(* IEC 61131-3 sources: MyTestRepos/BATTERY/PRG/BATTERY, 3 files *)

(* ---- PRG_Battery.st ---- *)
PROGRAM PRG_Battery
VAR
	ManualEnterPowerSaveMode: BOOL;	(*Manual Command to enter Power Save Mode for all packs*)
	ManualExitPowerSaveMode: BOOL;	(*Manual Command to exit Power Save Mode for all packs*)

	Extended_Statemachine: UINT := 0; (*Extended state machine for IAS, containing prewarning and shutdown  *)

	M : INT; (*Master of array information in Corvus BMS*)
	P : INT; (*Pack or packs with precharge module. Must receive connect command*)

	(*Battery Commands*)
	Connect: 				BOOL; (*Connect command from state machine*)
	Disconnect: 			BOOL; (*Disconnect command from state machine*)
	Tripstatus: 			DINT; (*Trip status from state machine*)
	ConnectPack1to8: 		DINT; (* Connect command read by communication programs*)
	testPrechargeTimeout: 	BOOL; (* Used to test precharge timeout *)
	ResetBattery : 			INT; (*Reset flag to Corvus BMS. 1 or 0 for true and false.*)
	CorvusConnect: 			fb_BitToWord; (*Split word to decide which packs to connect	*)

	(* Select and connect packs *)
	bms_Connect_Pack1: BOOL;
	bms_Select_Pack1: BOOL;
	bms_Connect_Pack2: BOOL;
	bms_Select_Pack2: BOOL;
	bms_Connect_Pack3: BOOL;
	bms_Select_Pack3: BOOL;
	bms_Connect_Pack4: BOOL;
	bms_Select_Pack4: BOOL;
	bms_Connect_Pack5: BOOL;
	bms_Select_Pack5: BOOL;
	bms_Connect_Pack6: BOOL;
	bms_Select_Pack6: BOOL;
	bms_Connect_Pack7: BOOL;
	bms_Select_Pack7: BOOL;
	bms_Connect_Pack8: BOOL;
	bms_Select_Pack8: BOOL;
	ConnectRS: RS;
	DeSelectTOF: TOF;

	(*Battery Feedback*)
	BatteryAllConnected: 	BOOL; (*All packs are connected*)
	BatteryMinOneConnected: BOOL; (*At least one pack is connected*)
	BatteryDisconnected : 	BOOL; (*All packs are disconnected*)
	BatteryReady: 			BOOL; (*Precharge pack is ready to connect or in power save mode*)
	BatteryConnecting: 		BOOL; (*Precharge pack is currently connecting*)
	BatteryReadyConnect:	BOOL; (*Battery is ready to connect or already connected or in power save mode - start sequence allowed*)

	(*Power Save Mode*)
	BatteryPackPowerSaveArray : 		ARRAY[1..16] OF INT; 	(*Count packs in power save mode*)
	BatteryCountPowerSave : 			DWORD;		(* Check how many packs are in power save mode*)
	BatteryNumInPowerSave : 			INT; 		(*Number of packs in power save mode*)
	BatteryAllPacksSleeping: 			BOOL; 		(*All battery packs are in power save mode*)
	ExitPowerSaveMode : 				BOOL;		(*Command to exit power save mode for all packs.*)
	GoToPowerSaveModeTP : 				TP;			(*Command Pulse*)
	ExitPowerSaveModeTP : 				TP;			(*Command Pulse*)
	LastPackDisconnectedRT: 			R_TRIG;		(*Rising edge trigger to detect when battery pack is no longer connected*)
	DelayPowerSaveAfterDisconnectTOF: 	TOF; 		(*Delay after last pack disconnect before entering power save mode*)
	DelayPowerSaveAfterDisconnectFT:	F_TRIG;		(*Falling edge trigger to enter power save when timer has run out*)
	EmergencyGoToPowerSaveRT: 			R_TRIG;		(*Detect when battery protection calls for emergency power save*)
	ForceSleepMode:						BOOL;		(*Bit from *)
	EnterPowerSaveModeTP:				TP;			(*Pulse to enable power save mode to Corvus*)
	AllowPowerSaveMode:					BOOL;		(*Power Save is only allowed for packs not in Connected eller Connecting State*)
	BatteriesInPowerSaveArray:			ARRAY[1..16] OF INT;	(*Array to register packs in power save mode*)
	BatteriesNotAllowedToSleepArray:	ARRAY[1..16] OF INT;	(*Array to register packs which are not allowed to sleep*)

	(*SoH Verification Testing*)
	SoHCurrent: 				INT := 0; (* Current limit during SoH Verification Testing*)

	(*Battery Charge/Discharge control*)
	StopDischargeTOF: 					TOF;					(*Discharge limit reached - limit discharge current to zero for some time*)
	StopChargeTOF: 						TOF;					(*Charge limit reached - limit charge current to zero for some time*)
	BMS_DischargeLimit_eng: 			DINT := 0;				(*Current limit in ampere*)
	BMS_ChargeLimit_eng: 				DINT := 0;				(*Current limit in ampere*)
	Battery_Current_Limiter: 	fb_CorvusOrcaCurrentLimiter;	(*Limitation function based on current*)
	ChargeLimitFilter:					FILTER_I;				(*Current filter used when stopping normally*)
	DischargeLimitFilter:				FILTER_I;				(*Current filter used when stopping normally*)
	ChargeLimit_eng: 					REAL := 0;				(* Charge limit in in ampere*)
	DischargeLimit_eng: 				REAL := 0;				(* Discharge limit in in ampere*)
	DriveDischargeLimit_eng: 			REAL := 0;				(* Discharge current in ampere used to limit DC/DC drive*)
	DriveChargeLimit_eng: 				REAL := 0;				(* Charge current in ampere used to limit DC/DC drive*)

	(*Readings and statuses*)
	SoC_Floor : INT; (*Current SoC level where the batteries are disconnected due to safety reasons / undervoltage*)
	busPower: REAL := 0; (* Power in kW to/from the batteries*)
	packSOH: ARRAY [1..16] OF REAL; (*Array of all pack's State of Health*)
	packSOC: ARRAY [1..16] OF REAL; (*Array of all pack's State of Charge*)

	MinutesRemaining: REAL := 0; (*Minutes remaining till current SoC_Floor, i.e. when batteries will auto disconnect. SoC Floor can vary depending on mode.*)
	hoursRemaining: REAL := 0; (*Hours remaining till current SoC_Floor, i.e. when batteries will auto disconnect. SoC Floor can vary depending on mode.*)
	energyRemaining: REAL := 0; (*Energy remaining on batteries in kWh*)
	energyRemainingOffline: REAL := 0; (*Energy in kWh remaining on batteries in offline mode. The lowest SoC is used.*)
	EnergyToFull: REAL := 0; (*Energy in kWh remaining until fully charged, SoC = 100% *)
	EnergyToDisconnect: REAL := 0; (*Energy in kWh remaining until completely discharged, SoC = 0% *)
	batteryCharging: BOOL; (*True if current is positive, i.e. current is flowing into the batteries*)

	(*Counter variables*)
	i:INT;
	y:INT;

	(*IAS Calculated variables*)
	avgCellVolt_sum: REAL := 0;
	avgCellTemp_sum: REAL := 0;
	AvailablePower : UINT;
	avgCellVolt : INT;
	avgCellTemp : INT;
	cellBalancingStatus : ARRAY[1..16] OF BOOL;
	CellsInBalance : ARRAY[1..16] OF BOOL;
	connectionArray : ARRAY[1..16] OF BOOL;
	AvailableEnergy : UINT;
END_VAR

(*
 * =======================================================================================================================================
 * Initial paper work; select Master and map commands from state machine
 * =======================================================================================================================================
*)

(*Decide which Corvus Controller to use as (M)aster for array data and (P)recharge/connect commands*)
M := PRG_BatteryComm.M;
P := PRG_BatteryComm.P;

(*Read commands from prg_Statemachine*)
Connect := PRG_StateMain.ConnectBattery ;
Disconnect := PRG_StateMain.DisconnectBattery ;
Tripstatus := PRG_StateMain.tripStatus ;

(*
 * =======================================================================================================================================
 * Connect and Disconnect Commands
 * =======================================================================================================================================
*)

(*RS function to hold connect command to Corvus.  *)
ConnectRS(SET := (Connect AND NOT testPrechargeTimeout), RESET1 := Disconnect OR (Tripstatus <> 0));

bms_Connect_Pack1 := (PRG_HMI.setup_Battery_total_nr_of_packs >= 1) AND ConnectRS.Q1;
bms_Connect_Pack2 := (PRG_HMI.setup_Battery_total_nr_of_packs >= 2) AND ConnectRS.Q1;
bms_Connect_Pack3 := (PRG_HMI.setup_Battery_total_nr_of_packs >= 3) AND ConnectRS.Q1;
bms_Connect_Pack4 := (PRG_HMI.setup_Battery_total_nr_of_packs >= 4) AND ConnectRS.Q1;
bms_Connect_Pack5 := (PRG_HMI.setup_Battery_total_nr_of_packs >= 5) AND ConnectRS.Q1;
bms_Connect_Pack6 := (PRG_HMI.setup_Battery_total_nr_of_packs >= 6) AND ConnectRS.Q1;
bms_Connect_Pack7 := (PRG_HMI.setup_Battery_total_nr_of_packs >= 7) AND ConnectRS.Q1;
bms_Connect_Pack8 := (PRG_HMI.setup_Battery_total_nr_of_packs >= 8) AND ConnectRS.Q1;

DeSelectTOF(
		IN := ConnectRS.Q1,
		PT := T#2500ms
);

(*Make sure packs are not de-selected prior to disconnect command*)
bms_Select_Pack1 := DeSelectTOF.Q;
bms_Select_Pack2 := DeSelectTOF.Q;
bms_Select_Pack3 := DeSelectTOF.Q;
bms_Select_Pack4 := DeSelectTOF.Q;
bms_Select_Pack5 := DeSelectTOF.Q;
bms_Select_Pack6 := DeSelectTOF.Q;
bms_Select_Pack7 := DeSelectTOF.Q;
bms_Select_Pack8 := DeSelectTOF.Q;

(*Prepare connection setup to Corvus*)
CorvusConnect(
	EN := TRUE,
	Bit0 := bms_Connect_Pack1,
	Bit1 := bms_Select_Pack1,
	Bit2 := bms_Connect_Pack2,
	Bit3 := bms_Select_Pack2,
	Bit4 := bms_Connect_Pack3,
	Bit5 := bms_Select_Pack3,
	Bit6 := bms_Connect_Pack4,
	Bit7 := bms_Select_Pack4,
	Bit8 := bms_Connect_Pack5,
	Bit9 := bms_Select_Pack5,
	Bit10 := bms_Connect_Pack6,
	Bit11 := bms_Select_Pack6,
	Bit12 := bms_Connect_Pack7,
	Bit13 := bms_Select_Pack7,
	Bit14 := bms_Connect_Pack8,
	Bit15 := bms_Select_Pack8,
	OUT => ConnectPack1to8
);

(*Battery is connected only when all packs are connected*)
BatteryAllConnected := (PRG_BatteryComm.CorvusRead[M].theArray.nrOfPackConnected = PRG_HMI.setup_Battery_total_nr_of_packs);

(*At least one pack is connected*)
BatteryMinOneConnected := (PRG_BatteryComm.CorvusRead[M].theArray.nrOfPackConnected >= 1);

(*Battery is disconnected only when all packs are disconnected*)
BatteryDisconnected := (PRG_BatteryComm.CorvusRead[M].theArray.nrOfPackConnected = 0);

(*Battery is ready when Pack controller with precharge is ready*)
BatteryReady := ((PRG_BatteryComm.CorvusRead[P].Pack.operationMode = 3) OR (PRG_BatteryComm.CorvusRead[P].Pack.operationMode = 1));

(*Connecting when precharge pack is working its magic*)
BatteryConnecting := (PRG_BatteryComm.CorvusRead[P].Pack.operationMode = 4);

(*Battery Ready to be Connected*)
BatteryReadyConnect := ((PRG_BatteryComm.CorvusRead[P].Pack.operationMode = 3) OR (PRG_BatteryComm.CorvusRead[P].Pack.operationMode = 5) OR (PRG_BatteryComm.CorvusRead[P].Pack.operationMode = 1));

(*
 * =======================================================================================================================================
 * Power Save Mode
 * =======================================================================================================================================
*)

(*Protection conditions to enter power save mode*)
EmergencyGoToPowerSaveRT(CLK := ForceSleepMode);

(*Enter power save mode when disconnect timer has run out*)
LastPackDisconnectedRT(
	CLK := (NOT BatteryMinOneConnected),
);

(*Enter power save mode when disconnect timer has run out*)
DelayPowerSaveAfterDisconnectTOF(
	IN := LastPackDisconnectedRT.Q,
	PT := REAL_TO_TIME(PRG_HMI.Delay_EnterPowerSaveMode*3600000)
);
DelayPowerSaveAfterDisconnectFT(CLK:=DelayPowerSaveAfterDisconnectTOF.Q);

EnterPowerSaveModeTP(
	IN := (DelayPowerSaveAfterDisconnectFT.Q OR ManualEnterPowerSaveMode OR EmergencyGoToPowerSaveRT.Q) AND PRG_HMI.enPowerSaveMode AND AllowPowerSaveMode,
	PT := T#2s,
	Q => (*Output is read in PRG_BatteryComm*),
	ET =>
);

(*Exit power save mode when starting*)
ExitPowerSaveModeTP(
	IN := PRG_Operation.ControlPlace.Start OR ManualExitPowerSaveMode,
	PT := T#2s,
	Q => ExitPowerSaveMode,
	ET =>
);

(*For loop to check how the batteries are sleeping or if they are allowed to go to sleep*)
FOR i:=1 TO PRG_HMI.setup_Battery_total_nr_of_packs BY 1 DO

	(*Check which batteries are in power save mode*)
	IF (PRG_BatteryComm.CorvusRead[i].Pack.operationMode = 1) THEN
		BatteriesInPowerSaveArray[i] := i*1;
	ELSE
		BatteriesInPowerSaveArray[i] := 0;
	END_IF

	(*Check which batteries are not allowed to enter power save*)
	IF (PRG_BatteryComm.CorvusRead[i].Pack.operationMode = 4 OR PRG_BatteryComm.CorvusRead[i].Pack.operationMode = 5) THEN
		BatteriesNotAllowedToSleepArray[i] := i*1;
	ELSE
		BatteriesNotAllowedToSleepArray[i] := 0;
	END_IF

END_FOR

(*Check how many battery packs are in power save mode*)
BatteryNumInPowerSave :=	BIT_COUNT(REAL_TO_DWORD((ARRAY_SUM(pt := ADR(BatteriesInPowerSaveArray), size := SIZEOF(BatteriesInPowerSaveArray)))));
IF (BatteryNumInPowerSave = PRG_HMI.setup_Battery_total_nr_of_packs) THEN
	BatteryAllPacksSleeping := TRUE;
ELSE
	BatteryAllPacksSleeping := FALSE;
END_IF

(*Power Save Mode is not allowed if any pack is either connected or connected*)
AllowPowerSaveMode := ( ARRAY_MAX(pt := ADR(BatteriesNotAllowedToSleepArray), size := SIZEOF(BatteriesNotAllowedToSleepArray))   <> 0);

(*
 * =======================================================================================================================================
 * Limitation of power to and from battery
 * =======================================================================================================================================
*)

(*------------------------------------- Batterilimiter fra BMS----------------------------------------------*)
(*This logic alters current limiters being sent into the limiter block. The output is filtered and controlled to vacon*)
IF (PRG_HMI.ChargeDischargeCurrentTestActive) THEN
	BMS_ChargeLimit_eng := LIMIT (0,REAL_TO_DINT(PRG_HMI.ChargeCurrentLimit_scale.PV),PRG_BatteryComm.CorvusRead[M].theArray.systemChargelimit);
	BMS_DischargeLimit_eng := LIMIT (0,REAL_TO_DINT(PRG_HMI.DischargeCurrentLimit_scale.PV),PRG_BatteryComm.CorvusRead[M].theArray.systemDischargeLimit);

ELSIF (PRG_HMI.SoHVerifModeActive) THEN (*Limit current to C-rate during State of Health Verification testing*)
	BMS_ChargeLimit_eng := LIMIT (0,INT_TO_DINT(SoHCurrent),PRG_BatteryComm.CorvusRead[M].theArray.systemChargelimit);
	BMS_DischargeLimit_eng := LIMIT (0,INT_TO_DINT(SoHCurrent),PRG_BatteryComm.CorvusRead[M].theArray.systemDischargeLimit);

ELSE
	BMS_ChargeLimit_eng := PRG_BatteryComm.CorvusRead[M].theArray.systemChargelimit;
	BMS_DischargeLimit_eng := PRG_BatteryComm.CorvusRead[M].theArray.systemDischargeLimit;
END_IF

(*Reading Charge/discharge limits and bus current in Ampere from BMS and compensates it by manipulating the reference*)
Battery_Current_Limiter(
	BMS_ChargeLimit_in := DINT_TO_INT(BMS_ChargeLimit_eng),
	BMS_DischargeLimit_in := DINT_TO_INT(BMS_DischargeLimit_eng),
	BatteryCurrent := PRG_BatteryComm.CorvusRead[M].theArray.busCurrent,
	NominalDriveCurrent := PRG_HMI.DriveSettings.SourceNomCurrent,
	BatteryConnected := BatteryMinOneConnected,
	ChargeLimit_eng => ,
	DischargeLimit_eng => ,
	ChargingLimited => ,
	DischargingLimited =>
);

(*Stop charging when battery voltage or SoC is too high*)
StopChargeTOF(
	IN := PRG_BatteryProtection.ChargeLimitWord <> 0,
	PT := T#30s, (*We want to stop charging for at least some time to prevent "blinking" of limits*)
	Q => ,
	ET =>
);

 (*Stop discharging when battery voltage or SoC is too low*)
StopDischargeTOF(
	IN:= PRG_BatteryProtection.DischargeLimitWord <> 0,
	PT := T#30s, (*We want to stop charging for at least some time to prevent "blinking" of limits*)
	Q => ,
	ET =>
);

(*Calculate charge/discharge limit from C-rate - Used as input to BMS Limiter during SoH verification*)
SoHCurrent := REAL_TO_INT(PRG_HMI.SoHChargeDischargeRate * setup_Battery_C_Rate * PRG_BatteryComm.CorvusRead[M].theArray.nrOfPackConnected);

(*This logic alters limits. Used for deloading or limiting when past SoC Low and Soc High*)

(*Ramping down limits towards zero to deload when stopping*)
IF ((PRG_StateMain.State = e_Stopping))  THEN
	ChargeLimit_eng := 0;
	DischargeLimit_eng := 0;

(*Limit when over charging - allowed to discharge*)
ELSIF (StopChargeTOF.Q) THEN
	ChargeLimit_eng := 0;
	DischargeLimit_eng := Battery_Current_Limiter.DischargeLimit_eng;

(*Limit when over discharging - allowed to charge*)
ELSIF (StopDischargeTOF.Q) THEN
	ChargeLimit_eng := Battery_Current_Limiter.ChargeLimit_eng;
	DischargeLimit_eng :=	0;

(*Normal operational limits controlled by BMS and other protective functions*)
ELSE
	ChargeLimit_eng := 		Battery_Current_Limiter.ChargeLimit_eng;
	DischargeLimit_eng := 	Battery_Current_Limiter.DischargeLimit_eng;
END_IF

(* Filtering of limit value*)
DischargeLimitFilter(
	X := REAL_TO_INT(DischargeLimit_eng),
	T := T#2s
);

ChargeLimitFilter(
	X := REAL_TO_INT(ChargeLimit_eng),
	T := T#2s
);

(*Preparing limit value to PRG_Drive*)
DriveChargeLimit_eng := 		ChargeLimitFilter.Y;
DriveDischargeLimit_eng := 		DischargeLimitFilter.Y;

(*
 * =======================================================================================================================================
 * Calculate Energy in batteries and time to full/empty/disconnect
 * =======================================================================================================================================
*)

(* Check if we are charging or discharging the battery *)
batteryCharging := (PRG_BatteryComm.CorvusRead[M].theArray.busPowerCalculated > 0 AND (PRG_BatteryComm.CorvusRead[M].Pack.operationMode = 5));

(*Calculate offline available energy, based on all packs and minimum state of charge*)
energyRemainingOffline := (
 	ARRAY_MIN(pt:=ADR(packSOC), size:=SIZEOF(packSOC)) *  	(* Lowest State of Charge *)
	setup_Energy_per_pack *									(* kWh per pack *)
	PRG_HMI.setup_Battery_total_nr_of_packs *				(* Total number of packs in array *)
	ARRAY_MIN(pt:=ADR(packSOH), size:=SIZEOF(packSOH)) *	(* Systems state of health *)
	0.0001													(* Correction factor *)
);

(*Calculate remaining energy to zero in an online system*)
EnergyToDisconnect := (
 	(PRG_BatteryComm.CorvusRead[M].theArray.systemOnlineSOC - REAL_TO_DINT(PRG_HMI.BMS_SoC.LL)) *  (* State of charge *)
	setup_Energy_per_pack *											(* kWh per pack *)
	PRG_BatteryComm.CorvusRead[M].theArray.nrOfPackConnected *		(* Number of packs online *)
	PRG_BatteryComm.CorvusRead[M].theArray.systemOnlineSOH *		(* Systems state of health *)
	0.0001															(* Correction factor *)
);

(*Calculate energy to full state of charge in an online system*)
EnergyToFull := (
 	setup_Energy_per_pack * 										(* kWh per pack *)
 	PRG_BatteryComm.CorvusRead[M].theArray.nrOfPackConnected *		(* Number of packs online *)
	PRG_BatteryComm.CorvusRead[M].theArray.systemOnlineSOH *		(* Systems state of health *)
	0.01															(* Correction factor *)
) - EnergyToDisconnect;												(* Subtract remaining energy *)

(*Prevent division by zero when calculating time remaining (This result is the denominator in the energy division) *)
IF PRG_BatteryComm.CorvusRead[M].theArray.busPowerCalculated = 0
	THEN busPower := 0.1;
	ELSE busPower := PRG_BatteryComm.CorvusRead[M].theArray.busPowerCalculated;
END_IF

(* Calculate time remaining to either 100% or 0% depending on whether the battery is charging or discharging *)
IF (batteryCharging) THEN
	hoursRemaining := EnergyToFull/busPower;
ELSE
	hoursRemaining := EnergyToDisconnect/busPower;
END_IF

MinutesRemaining := ABS(hoursRemaining*60);

(*
 * =======================================================================================================================================
 * Calculate values for IAS information
 * =======================================================================================================================================
*)

FOR i:=1 TO 16 BY 1 DO

	(*Set up all pack state of charges in an array*)
	IF ((PRG_BatteryComm.CorvusRead[i].Pack.SOC <> 0) OR PRG_BatteryComm.CorvusRead[i].ModbusFault) THEN
		packSOC[i] := DINT_TO_REAL(PRG_BatteryComm.CorvusRead[i].Pack.SOC);
	ELSE
		packSOC[i] := 999; (*prevent zeros in array when looking for the lowest value*)
	END_IF

	(*Set up all pack state of health in an array*)
	IF ((PRG_BatteryComm.CorvusRead[i].Pack.SOH <> 0) OR PRG_BatteryComm.CorvusRead[i].ModbusFault) THEN
		packSOH[i] := DINT_TO_REAL(PRG_BatteryComm.CorvusRead[i].Pack.SOH);
	ELSE
		packSOH[i] := 999; (*prevent zeros in array when looking for the lowest value*)
	END_IF

	(*Count pack balancing status*)
	IF (PRG_BatteryComm.CorvusRead[i].Pack.cellBalancingStatus = 1) THEN
		cellBalancingStatus[i] :=  TRUE;
	ELSE
		cellBalancingStatus[i] :=  FALSE;
	END_IF;

	(*Count pack balancing status 2*)
	IF (PRG_BatteryComm.CorvusRead[i].Pack.cellsInBalance = 1) THEN
		CellsInBalance[i] :=  TRUE;
	ELSE
		CellsInBalance[i] :=  FALSE;
	END_IF;

	(*Connection Array*)
	IF (PRG_BatteryComm.CorvusRead[i].Pack.operationMode = 5) THEN
		connectionArray[i] :=  TRUE;
	ELSE
		connectionArray[i] :=  FALSE;
	END_IF;
END_FOR

(*Find average cell temperature*)
avgCellTemp_sum := 0;
FOR i:=1 TO PRG_HMI.setup_Battery_total_nr_of_packs BY 1 DO
	avgCellTemp_sum := avgCellTemp_sum + DINT_TO_REAL(PRG_BatteryComm.CorvusRead[i].Pack.avgCellTemp);
END_FOR
avgCellTemp := REAL_TO_INT(fun_SafeDivide(divident := avgCellTemp_sum, devisor := PRG_HMI.setup_Battery_total_nr_of_packs));

(*Find average cell voltage*)
avgCellVolt_sum := 0;
FOR i:=1 TO PRG_HMI.setup_Battery_total_nr_of_packs BY 1 DO
	avgCellVolt_sum := avgCellVolt_sum + DINT_TO_REAL(PRG_BatteryComm.CorvusRead[i].Pack.avgCellVoltage);
END_FOR
avgCellVolt := REAL_TO_INT(fun_SafeDivide(divident := avgCellVolt_sum, devisor := PRG_HMI.setup_Battery_total_nr_of_packs));

(*Determine wether to use online or offline energy*)
IF (PRG_BatteryComm.CorvusRead[M].theArray.nrOfPackConnected > 0) THEN
	AvailableEnergy := REAL_TO_UINT(EnergyToDisconnect);
ELSE
	AvailableEnergy := REAL_TO_UINT(energyRemainingOffline);
END_IF

(*Send offline estimated available power to IAS/PMS*)
IF (PRG_BatteryComm.CorvusRead[M].theArray.nrOfPackConnected > 0) THEN
	AvailablePower := REAL_TO_UINT( MIN(PRG_BatteryComm.CorvusRead[M].theArray.systemDischargeLimit,PRG_HMI.DriveSettings.SourceNomCurrent) * PRG_BatteryComm.CorvusRead[M].theArray.busVoltage/1000);
ELSE
	AvailablePower := REAL_TO_UINT((PRG_HMI.DriveSettings.SourceNomCurrent * PRG_BatteryComm.CorvusRead[M].Pack.batteryVoltage)/1000);
END_IF

(* IAS extended state machine status containing prewarning and shutdown *)
IF (PRG_BatteryProtection.batteryPreWarning AND NOT (PRG_StateMain.tripStatus <> 0)) THEN
	Extended_Statemachine := 6;
ELSIF (PRG_StateMain.tripStatus <> 0) THEN
	Extended_Statemachine := 7;
ELSE
	Extended_Statemachine := PRG_StateMain.State;;
END_IF

END_PROGRAM

ACTIONS

END_ACTIONS

(* ---- PRG_BatteryComm.st ---- *)
(*
 * This program instantiates the Corvus Orca communication function block and gathers write-commands from other programs.
 * Made by: YS
 * Last changed: 2018-09-18
*)
PROGRAM PRG_BatteryComm

VAR
	mb_BMS_arrayData: 	ARRAY [1..16] OF str_Corvus_Array; 		(*Almighty array containing all information about PV and alarms for analog input signals*)
	mb_BMS_packData: 	ARRAY [1..16] OF str_Corvus_packData;	(*Almighty array containing all information about PV and alarms for analog input signals*)
	mb_BMS_packFW: 		ARRAY [1..16] OF str_Corvus_packFW; 	(*Almighty array containing all information about PV and alarms for analog input signals*)
    CorvusRead: 		ARRAY [1..16] OF str_Corvus_ALL; 		(*The almighty Corvus BMS Array-Array*)
	CorvusWrite: 		ARRAY [1..16] OF str_Corvus_Write;		(*Command Register Array to Corvus pack controllers*)

	CorvusModbusFault_TON: 				TON;							(*Timer to declare modbus communication fault*)
	Modbus_Wait:						BOOL;							(*Start to wait before restarting modbus fault checking*)
	Modbus_WaitRT:						R_TRIG;							(*Puls detection to start timer*)
	Modbus_WaitTryFT:					F_TRIG;							(*Puls detection that timer has ended*)
	ModbusFault_WaitTry_TP:				TP;								(*Timer to wait before restarting check of array*)
	CorvusBMS_Total_Comm_Fault_SR:		SR;								(*The Total Modbus Fault must be latched unntil we know it is healthy again*)
	CorvusBMS_Reset_Total_Comm_Fault_TON:TON;							(*Wait this long before declaring that communication is OK again*)
	NoPrechargePackComm: 				BOOL; 							(*Alarm when there is modbus fault on all packs which can start/stop*)
	n: 									INT := 0; 						(*Looping variable for reset function*)
	i: 									INT; 							(*Looping variable for checking comm fault across packs*)
	M : 								INT:=1; 						(*Pack number for current Array Master: The pack that array information is gathered from*)
	P : 								INT:=1; 						(*Pack number for current Array Precharge Master: The pack that can initiate start/connect requests*)
	Corvus_Array : 						fb_CorvusOrcaComm; 				(*All corvus data*)
	WriteCommands : 					ARRAY[1..16] OF str_Corvus_Write; (*Command Register Array to Corvus pack controllers*)

	(*Commands read from other programs*)
	Reset : 							BOOL; 							(*Reset command for battery packs*)
	CorvusBMS_Total_Comm_Fault_TON : 	TON;
	CorvusBMS_Total_Comm_Fault: 		BOOL; 							(*No communication with any Corvus batteries :( *)

	(*Variables to HMI*)
	setup_AlarmDelay_Modbus : 			TIME:=T#5s;		(*Delay before issuing total comm failure alarm*)
END_VAR

Reset := PRG_Functions.Reset;

(*
 * =======================================================================================================================================
 * Communication with Corvus Orca Battery Management
 * =======================================================================================================================================
*)
Corvus_Array(
 	First_Card_ID:=PRG_HMI.setup_Battery_First_Card_Nr,
 	Number_of_packs_in_array:=PRG_HMI.setup_Battery_total_nr_of_packs ,
 	corvusWrite := WriteCommands,
 	Reset := Reset,
 	output => CorvusRead
);

(*
 * =======================================================================================================================================
 * Find Array Master (M) - This is the array we use most data from
 * =======================================================================================================================================
*)

IF CorvusRead[M].ModbusFault AND CorvusRead[1].ModbusFault AND  M<= PRG_HMI.setup_Battery_total_nr_of_packs AND NOT ModbusFault_WaitTry_TP.Q  THEN
	(*If current array master and pack 1 has comm fault, try next one as long as we still have more packs in the array to try*)
	M := M+1;
	Modbus_Wait := FALSE;
ELSIF M > PRG_HMI.setup_Battery_total_nr_of_packs OR NOT CorvusRead[1].ModbusFault THEN
	(*If array 1 is ok *OR* there are no more arrays to try - go for number 1*)
	M := 1;
	Modbus_Wait := TRUE;	(*After running through all arrays, wait before restarting so that CorvusBMS_Total_Comm_Fault_TON can detect that we have no-one to talk to*)
END_IF

Modbus_WaitRT(CLK := Modbus_Wait); (*Create an R_trig to start the TP*)
ModbusFault_WaitTry_TP(				(*When we have tested all arrays and found no-one to communicate with, take a pause before re-starting so that we can detect the comm fault*)
		IN := Modbus_WaitRT.Q,
		PT := setup_AlarmDelay_Modbus + INT_TO_TIME(1000) (*Make sure that the re-try delay is longer than the alarm delay. 1000 = 1 s *)
	);
Modbus_WaitTryFT(CLK := ModbusFault_WaitTry_TP.Q); (*Detect when the pause is finished so that the pause-command can be turned off*)

IF(Modbus_WaitTryFT.Q OR NOT CorvusRead[M].ModbusFault) THEN
	Modbus_Wait := FALSE;
END_IF

(*No success in finding an Array master without communication fault - issue alarm*)
CorvusBMS_Total_Comm_Fault_TON(
	IN := CorvusRead[M].ModbusFault,
	PT := setup_AlarmDelay_Modbus
);

(*Make sure that the re-established communication is stable before clearing the alarm*)
CorvusBMS_Reset_Total_Comm_Fault_TON(
	IN := NOT Modbus_Wait,
	PT := setup_AlarmDelay_Modbus + INT_TO_TIME(2000), (*The "stable time" must be longer than the pause between retry-attemps*)
	Q => ,
	ET =>
);

(*Latch the modbus fault and reset it when communication has been restored for a time*)
CorvusBMS_Total_Comm_Fault_SR(
	SET1 := CorvusBMS_Total_Comm_Fault_TON.Q,
	RESET := CorvusBMS_Reset_Total_Comm_Fault_TON.Q OR PRG_Functions.Reset,
	Q1 => CorvusBMS_Total_Comm_Fault
);

(*
 * =======================================================================================================================================
 * Find Array Precharge Master (P) - This is the array we send start commands to
 * =======================================================================================================================================
*)

IF NOT CorvusRead[setup_Battery_PrechargePackA].ModbusFault THEN
	(*If pack A is home sick but pack B is ok - it's all good*)
	P := setup_Battery_PrechargePackA;
	NoPrechargePackComm := FALSE;
ELSE
	NoPrechargePackComm := TRUE;
END_IF

(*
 * =======================================================================================================================================
 * Write Commands
 * =======================================================================================================================================
*)

(*Connect Commands*)
WriteCommands[M].connectPack1to8 := PRG_Battery.ConnectPack1to8;

(*Power Save Commands*)
IF (PRG_Battery.EnterPowerSaveModeTP.Q) THEN
	WriteCommands[M].systemPowerSaveControl := 2;
ELSIF (PRG_Battery.ExitPowerSaveModeTP.Q) THEN
	WriteCommands[M].systemPowerSaveControl := 3;
ELSE
	WriteCommands[M].systemPowerSaveControl := 0;
END_IF

(* Reset all pack controllers *)
IF (Reset AND CorvusRead[M].theArray.nrOfPackFault > 0) THEN
	FOR n := 1 TO PRG_HMI.setup_Battery_total_nr_of_packs BY 1 DO
		WriteCommands[n].systemAlarmReset := 1;
	END_FOR
	n := 1;
ELSIF(Reset AND CorvusRead[M].theArray.nrOfPackFault = 0) THEN
	FOR n := 1 TO PRG_HMI.setup_Battery_total_nr_of_packs BY 1 DO
		WriteCommands[n].systemAlarmReset := 0;
	END_FOR
	n := 1;
ELSIF(NOT Reset) THEN
	FOR n := 1 TO PRG_HMI.setup_Battery_total_nr_of_packs BY 1 DO
		WriteCommands[n].systemAlarmReset := 0;
	END_FOR
	n := 1;
END_IF

;
END_PROGRAM

ACTIONS

END_ACTIONS

(* ---- PRG_BatteryProtection.st ---- *)
PROGRAM PRG_BatteryProtection
VAR
	(* Find any BMS Array warning associated with a pre-warning*)
	batteryPreWarning: 			BOOL; 					(*True if any pack has one or more prewarning alarms*)
	BatteryPreWarnings_Array: 	ARRAY[1..16] OF INT; 	(*Array to gather information about prewarning alarms from all packs*)

	(*Find any common warning from the battery array*)
	batteryCommonWarning: 		BOOL; 					(*True if any pack has one or more warnings*)
	BatteryWarnings_Array: 		ARRAY[1..16] OF INT; 	(*Array to gather information about warning alarms from all packs*)

	(*Find any common fault from the battery array*)
	batteryCommonFault: 		BOOL; (*True if any pack has an active/unacknowledged fault*)

	(*Common Faults from Battery Array*)
	Common_SE_overVoltage_Fault_Array: 					ARRAY[1..16] OF INT; (*Array of BOOLs from BMS: *)
	Common_SE_underVoltage_Fault_Array: 				ARRAY[1..16] OF INT; (*Array of BOOLs from BMS: *)
	Common_SE_overTemperature_Fault_Array: 				ARRAY[1..16] OF INT; (*Array of BOOLs from BMS: *)
	Common_HVIL_Fault_Array: 							ARRAY[1..16] OF INT; (*Array of BOOLs from BMS: *)
	Common_E_Stop_Active_Fault_Array: 					ARRAY[1..16] OF INT; (*Array of BOOLs from BMS: *)
	Common_Safety_Shutdown_Fault_Array: 				ARRAY[1..16] OF INT; (*Array of BOOLs from BMS: *)
	Common_Ground_Fault_Fault_Array: 					ARRAY[1..16] OF INT; (*Array of BOOLs from BMS: *)
	Common_Contactor_Fault_Array: 						ARRAY[1..16] OF INT; (*Array of BOOLs from BMS: *)
	Common_Low_Temp_OverCurrent_Fault_Array: 			ARRAY[1..16] OF INT; (*Array of BOOLs from BMS: *)
	Common_Repeated_OverCharge_Lockout_Fault_Array: 	ARRAY[1..16] OF INT; (*Array of BOOLs from BMS: *)
	Common_Deep_OverDischarge_Lockout_Fault_Array: 		ARRAY[1..16] OF INT; (*Array of BOOLs from BMS: *)
	Common_PDM_OverTemperature_Fault_Array: 			ARRAY[1..16] OF INT; (*Array of BOOLs from BMS: *)

	Common_SE_overVoltage_Fault: 				BOOL; (*Any pack has a Cell Over Voltage Fault*)
	Common_SE_underVoltage_Fault: 				BOOL; (*Any pack has a Cell Under Voltage Fault*)
	Common_SE_overTemperature_Fault: 			BOOL; (*Any pack has a Cell Over Temperature Fault*)
	Common_HVIL_Fault: 							BOOL; (*Any pack has a High Voltage Interlock Loop fault*)
	Common_E_Stop_Active_Fault: 				BOOL; (*Any pack has a Emergency Stop Active Fault*)
	Common_Safety_Shutdown_Fault: 				BOOL; (*Any pack has a Safety Shutdown Fault*)
	Common_Ground_Fault_Fault: 					BOOL; (*Any pack has a Ground Fault*)
	Common_Contactor_Fault: 					BOOL; (*Any pack has a Contactor Fault*)
	Common_Low_Temp_OverCurrent_Fault: 			BOOL; (*Any pack has a Low Temperature Over Current Fault*)
	Common_Repeated_OverCharge_Lockout_Fault: 	BOOL; (*Any pack has a Repeated Over Charge Lockout Fault*)
	Common_Deep_OverDischarge_Lockout_Fault: 	BOOL; (*Any pack has a Common Deep Over Discharge Lockout Fault*)
	Common_PDM_OverTemperature_Fault: 			BOOL; (*Any pack has a Power Distribution Module Over Temperature Fault*)

	(*Common Warnings from Battery Array*)
	Common_SE_overVoltage_Warning_Array: 		ARRAY[1..16] OF INT; (*Array of BOOLs from BMS: *)
	Common_SE_underVoltage_Warning_Array: 		ARRAY[1..16] OF INT; (*Array of BOOLs from BMS: *)
	Common_SE_overTemperature_Warning_Array: 	ARRAY[1..16] OF INT; (*Array of BOOLs from BMS: *)
	Common_Module_Communication_Warning_Array: 	ARRAY[1..16] OF INT; (*Array of BOOLs from BMS: *)
	Common_OverCurrent_Warning_Array: 			ARRAY[1..16] OF INT; (*Array of BOOLs from BMS: *)
	Common_Input_PowerLoss_Warning_Array: 		ARRAY[1..16] OF INT; (*Array of BOOLs from BMS: *)
	Common_PDM_overTemperature_Warning_Array: 	ARRAY[1..16] OF INT; (*Array of BOOLs from BMS: *)
	Common_CoolantLeak_Warning_Array: 			ARRAY[1..16] OF INT; (*Array of BOOLs from BMS: *)
	Common_SE_overVoltage_Warning: 				BOOL; (*Any pack has a Common Cell Over Voltage Warning*)
	Common_SE_underVoltage_Warning: 			BOOL; (*Any pack has a Common Cell Under Voltage Warning*)
	Common_SE_overTemperature_Warning: 			BOOL; (*Any pack has a Common Cell Over Temperature Warning*)
	Common_Module_Communication_Warning: 		BOOL; (*Any pack has a Common Module Communication Warning*)
	Common_OverCurrent_Warning: 				BOOL; (*Any pack has a Common Over Current Warning*)
	Common_Input_PowerLoss_Warning: 			BOOL; (*Any pack has a Common Input Powerloss Warning*)
	Common_PDM_overTemperature_Warning: 		BOOL; (*Any pack has a Common Power Distribution Module Over Temperature Warning*)
	Common_CoolantLeak_Warning: 				BOOL; (*Any pack has a Common Coolant Water Leakage Warning*)

	CorvusRead: 			ARRAY [1..16] OF str_Corvus_ALL; (*The almighty Corvus BMS Array-Array*)
	BatteryAlone :			BOOL; 			(*If battery is alone, lower SoC trip limit is decreased*)
	BatteryCharging:	 	BOOL;			(*If battery is charging, discharging is still allowed beyond limits*)
	ConfigError:			INT;			(*Check that all protection settings are within hardcoded limits*)

	TripBasket : 			fb_16DelayedSR;	(*Collection basket for protection trips*)
	WarningBasket :			fb_16DelayedSR; (*Collection basket for warnings*)
	ProtectionTrip: 		DINT;			(*All bits from protection trips*)
	ChargeLimitWord :		WORD;			(*Word with bit-conditions for stop charging*)
	DischargeLimitWord :	WORD;			(*Word with bit-conditions for stop discharging*)

	Warning_SoC_L : 				BOOL;	(*Warning or trip bit*)
	Warning_SoC_L_Offline :			BOOL;	(*Warning or trip bit*)
	Warning_SoC_LL_Offline :		BOOL;	(*Warning or trip bit*)
	Warning_SoC_H : 				BOOL;	(*Warning or trip bit*)
	Warning_Volt_L : 				BOOL;	(*Warning or trip bit*)
	Warning_Volt_H : 				BOOL;	(*Warning or trip bit*)
	Warning_CellVolt_H :			BOOL;	(*Warning or trip bit*)
	Warning_CellVolt_L :			BOOL;	(*Warning or trip bit*)
	Warning_CellVolt_L_Offline :	BOOL;	(*Warning or trip bit*)
	Warning_CellVolt_LL_Offline :	BOOL;	(*Warning or trip bit*)
	Warning_CellTemp_H :			BOOL;	(*Warning or trip bit*)
	Warning_CellTemp_L :			BOOL;	(*Warning or trip bit*)
	Warning_BattRoomTemp_HH:		BOOL;	(*Warning or trip bit*)
	Warning_BattRoomTemp_H:			BOOL;	(*Warning or trip bit*)
	Warning_BattRoomTemp_L:			BOOL;	(*Warning or trip bit*)
	Warning_BattRoomTemp_LL:		BOOL;	(*Warning or trip bit*)

	ProtectionTrip_SoC_HH: 			BOOL;	(*Warning or trip bit*)
	ProtectionTrip_SoC_LL: 			BOOL;	(*Warning or trip bit*)
	ProtectionTrip_SoC_LLL: 		BOOL;	(*Warning or trip bit*)
	ProtectionTrip_CellTemp_HH:		BOOL;	(*Warning or trip bit*)
	ProtectionTrip_CellVolt_HH:		BOOL;	(*Warning or trip bit*)
	ProtectionTrip_CellVolt_LL:		BOOL;	(*Warning or trip bit*)
	ProtectionTrip_Overvoltage: 	BOOL;	(*Warning or trip bit*)
	ProtectionTrip_Undervoltage: 	BOOL;	(*Warning or trip bit*)
	M:INT;

	(*Offline Protection*)
	ForceSleepMode :		BOOL;					(*Conditions are so that we want to force batteries to sleep*)
	i: 						INT;					(*Looping variable*)
	minCellVoltage: 		REAL := 0;				(*The lowest cell voltage in the array*)
	minCellVoltageArray: 	ARRAY[1..16] OF REAL;	(*Array of lowest cell voltages in battery packs*)
	maxCellVoltage: 		REAL := 0;				(*The highest cell voltage in the array*)
	maxCellVoltageArray: 	ARRAY[1..16] OF REAL;	(*Array of highest cell voltages in battery packs*)

	minCellTemp: 			REAL := 0;				(*The lowest cell temperature in the array*)
	minCellTempArray: 		ARRAY[1..16] OF REAL;	(*Array of lowest cell temperature in battery packs*)
	maxCellTemp: 			REAL := 0;				(*The highest cell temperature in the array*)
	maxCellTempArray: 		ARRAY[1..16] OF REAL;	(*Array of highest cell temperature in battery packs*)

	minPackSoC: 			REAL := 0;				(*The lowest pack state of charge in the array*)
	minPackSoCArray: 		ARRAY[1..16] OF REAL;	(*Array of lowest pack state of charge in battery arrays*)
	maxPackSoC: 			REAL := 0;				(*The highest pack state of charge in the array*)
	maxPackSoCArray: 		ARRAY[1..16] OF REAL;	(*Array of highest pack state of charge in battery arrays*)
END_VAR

(*Read variables from other programs*)
CorvusRead :=		PRG_BatteryComm.CorvusRead;
M := 				PRG_BatteryComm.M;
BatteryCharging := 	PRG_Battery.batteryCharging;

(*BatteryAlone signal from PMS - SoC LL Trip is lowered to minimum*)
BatteryAlone := PRG_IAS.IAS_BatteryAlone;

(*Make sure that limits are within allowed values to exit init state in prg_StateMain*)
ConfigError.0 :=	(PRG_HMI.SetupBatLimits.SoCTripHH > setup_SoC_HH_Trip);
ConfigError.1 :=	(PRG_HMI.SetupBatLimits.SoCTripLL < setup_SoC_LLL_Trip);
ConfigError.2 :=	(PRG_HMI.SetupBatLimits.VoltTripHH > setup_Battery_Max_Voltage);
ConfigError.3 :=	(PRG_HMI.SetupBatLimits.VoltTripLL < setup_Battery_Min_Voltage);
ConfigError.4 :=	(PRG_HMI.SetupBatLimits.CellVoltTripHH > setup_Battery_CellVolt_HH_Trip);
ConfigError.5 :=	(PRG_HMI.SetupBatLimits.CellVoltTripLL < setup_Battery_CellVolt_LL_Trip);
ConfigError.6 :=	(PRG_HMI.SetupBatLimits.SoCTripLL_Offline < setup_Battery_SoC_Offline_LL_Trip);
ConfigError.7 :=	(PRG_HMI.SetupBatLimits.CellVoltTripLL_Offline < setup_Battery_CellVolt_Offline_LL_Trip);
ConfigError.8 :=	(PRG_HMI.SetupBatLimits.CellTempTripHH > setup_Battery_CellTemp_HH_Trip);
ConfigError.9 :=	FALSE;
ConfigError.10 :=	FALSE;
ConfigError.11 :=	FALSE;
ConfigError.12 :=	FALSE;
ConfigError.13 :=	FALSE;
ConfigError.14 :=	FALSE;
ConfigError.15 :=	FALSE;

ChargeLimitWord.0 := 	CorvusRead[M].theArray.systemOnlineSOC	> 	PRG_HMI.SetupBatLimits.SoCAlarmH;
ChargeLimitWord.1 := 	CorvusRead[M].theArray.maxCellVoltage	> 	PRG_HMI.SetupBatLimits.CellVoltAlarmH;
ChargeLimitWord.2 := 	CorvusRead[M].theArray.busVoltage 		> 	PRG_HMI.SetupBatLimits.VoltAlarmH;
ChargeLimitWord.3 := 	CorvusRead[M].theArray.systemOnlineSOC 	> 	PRG_HMI.SetupBatLimits.SoCAlarmH;

DischargeLimitWord.0 := (CorvusRead[M].theArray.systemOnlineSOC < 	PRG_HMI.SetupBatLimits.SoCAlarmL) 		AND PRG_Battery.BatteryMinOneConnected AND NOT BatteryAlone AND NOT (PRG_StateMain.State = e_Stopping);
DischargeLimitWord.1 :=	(CorvusRead[M].theArray.minCellVoltage 	< 	PRG_HMI.SetupBatLimits.CellVoltAlarmL) AND PRG_Battery.BatteryMinOneConnected AND NOT BatteryAlone AND NOT (PRG_StateMain.State = e_Stopping);
DischargeLimitWord.2 := (CorvusRead[M].theArray.busVoltage 		< 	PRG_HMI.SetupBatLimits.VoltAlarmL) 	AND PRG_Battery.BatteryMinOneConnected AND NOT BatteryAlone AND NOT (PRG_StateMain.State = e_Stopping);

(*All faults are collected here with individual time delay and latched output*)
TripBasket(

 	(* Prevent over SoC when charging *)
	in1 := ((CorvusRead[M].theArray.systemOnlineSOC > PRG_HMI.SetupBatLimits.SoCTripHH)
	 		AND (PRG_BatteryComm.CorvusRead[M].theArray.busPowerCalculated > -50) (*must be more than 50 kW discharging power before cancelling trip timer*)
	),
	delay1 := T#30s,
	out1 => ProtectionTrip_SoC_HH,

	(* Prevent Under SoC when discharging and there are other power sources on the switchboard *)
	in2 := ((CorvusRead[M].theArray.systemOnlineSOC < PRG_HMI.SetupBatLimits.SoCTripLL)
			AND NOT BatteryCharging
	 		AND PRG_Battery.BatteryMinOneConnected
	 		AND NOT BatteryAlone
	),
	delay2 := T#30s,
	out2 => ProtectionTrip_SoC_LL,

	(* Prevent Under SoC when discharging*)
	in3 := ((CorvusRead[M].theArray.systemOnlineSOC < PRG_HMI.SetupBatLimits.SoCTripLL)
	 		AND PRG_Battery.BatteryMinOneConnected
	 		AND (PRG_BatteryComm.CorvusRead[M].theArray.busPowerCalculated < 50) (*must be more than 50 kW charging power before cancelling trip timer*)
	),
	delay3 := T#30s,
	out3 => ProtectionTrip_SoC_LLL,

	(*Over Voltage Trip*)
	in4 := ((CorvusRead[M].theArray.busVoltage > PRG_HMI.SetupBatLimits.VoltTripHH)
	 		AND BatteryCharging
	),
	delay4 := T#30s,
	out4 => ProtectionTrip_Overvoltage,

	(*Under Voltage Trip*)
	in5 := ((CorvusRead[M].theArray.busVoltage < PRG_HMI.SetupBatLimits.VoltTripLL)
	 		AND NOT BatteryCharging
			AND  PRG_Battery.BatteryMinOneConnected
	),
	delay5 := T#30s,
	out5 => ProtectionTrip_Undervoltage,

	(*Cell over voltage trip*)
	in6 := (maxCellVoltage > PRG_HMI.SetupBatLimits.CellVoltTripHH
	 		AND PRG_Battery.BatteryMinOneConnected
	),
	delay6 := T#30s,
	out6 => ProtectionTrip_CellVolt_HH,

	(*Cell under voltage trip*)
	in7 := ((minCellVoltage < PRG_HMI.SetupBatLimits.CellVoltTripLL)
			AND NOT BatteryCharging
			AND  PRG_Battery.BatteryMinOneConnected
	),
	delay7 := T#30s,
	out7 => ProtectionTrip_CellVolt_LL,

	(*Cell over temperature trip*)
	in8 := (maxCellTemp > PRG_HMI.SetupBatLimits.CellTempTripHH
	 		AND PRG_Battery.BatteryMinOneConnected),
	delay8 := T#30s,
	out8 => ProtectionTrip_CellTemp_HH,

	in9 := FALSE,
	delay9 := T#0s,
	out9 => ,

	in10 := FALSE,
	delay10 := T#0s,
	out10 => ,

	in11 := FALSE,
	delay11 := T#0s,
	out11 => ,

	in12 := FALSE,
	delay12 := T#0s,
	out12 => ,

	in13 := FALSE,
	delay13 := T#0s,
	out13 => ,

	in14 := FALSE,
	delay14 := T#0s,
	out14 => ,

	in15 := FALSE,
	delay15 := T#0s,
	out15 => ,

	in16 := FALSE,
	delay16 := T#0s,
	out16 => ,

	Reset := PRG_Functions.Reset,
	outCommon => ProtectionTrip
);

(*All warnings are collected here with individual time delay and latched output*)
WarningBasket(

 	(*Low State of Charge Warning*)
	in1 := (CorvusRead[M].theArray.systemOnlineSOC < PRG_HMI.SetupBatLimits.SoCAlarmL)
			AND (CorvusRead[M].theArray.nrOfPackConnected > 0),
	delay1 := T#5s,
	out1 => Warning_SoC_L,

	(*High State of Charge Warning*)
	in2 := (CorvusRead[M].theArray.systemOnlineSOC > PRG_HMI.SetupBatLimits.SoCAlarmH),
	delay2 := T#5s,
	out2 => Warning_SoC_H,

	(*Low Battery Voltage Warning*)
	in3 := (CorvusRead[M].theArray.busVoltage < PRG_HMI.SetupBatLimits.VoltAlarmL)
			AND (CorvusRead[M].theArray.nrOfPackConnected > 0),
	delay3 := T#5s,
	out3 => Warning_Volt_L,

	(*High Battery Voltage Warning*)
	in4 := CorvusRead[M].theArray.busVoltage > PRG_HMI.SetupBatLimits.VoltAlarmH,
	delay4 := T#5s,
	out4 => Warning_Volt_H,

	(*High Cell Voltage*)
	in5 := maxCellVoltage > PRG_HMI.SetupBatLimits.CellVoltAlarmH,
	delay5 := T#5s,
	out5 => Warning_CellVolt_H,

	(*High Cell Temperature*)
	in6 := maxCellTemp > PRG_HMI.SetupBatLimits.CellTempAlarmH,
	delay6 := T#5s,
	out6 => Warning_CellTemp_H,

	(*Low Cell Voltage*)
	in7 := ((minCellVoltage < PRG_HMI.SetupBatLimits.CellVoltAlarmL)
	 			AND (minCellVoltage <> 0) (*We don't believe in zero values*)
	 			AND NOT PRG_BatteryComm.CorvusBMS_Total_Comm_Fault
	),
	delay7 := T#5s,
	out7 => Warning_CellVolt_L,

	(*Low Cell Temperature*)
	in8 := ((minCellTemp < PRG_HMI.SetupBatLimits.CellTempAlarmL)
	 			AND (minCellTemp <> 0) (*Zero might be plausible here, but if it is real it has nonetheless triggered the alarm when passing the limit on its way down*)
	 			AND NOT PRG_BatteryComm.CorvusBMS_Total_Comm_Fault
	),
	delay8 := T#5s,
	out8 => Warning_CellTemp_L,

	(*OFFLINE: Low SoC*)
	in9 := ((minPackSoC < PRG_HMI.SetupBatLimits.SoCAlarmL_Offline)
	 			AND NOT PRG_BatteryComm.CorvusBMS_Total_Comm_Fault
	),
	delay9 := T#5s,
	out9 => Warning_SoC_L_Offline,

	(*OFFLINE: Low Cell Voltage*)
	in10 := ((minCellVoltage < PRG_HMI.SetupBatLimits.CellVoltAlarmL_Offline)
	 			AND (minCellVoltage <> 0)  (*We don't believe in zero values*)
	 			AND NOT PRG_BatteryComm.CorvusBMS_Total_Comm_Fault
	),
	delay10 := T#5s,
	out10 => Warning_CellVolt_L_Offline,

	(*OFFLINE: Low Low Cell Voltage*)
	in11 := ((minCellVoltage < PRG_HMI.SetupBatLimits.CellVoltTripLL_Offline)
	 			AND (minCellVoltage <> 0)  (*We don't believe in zero values*)
	 			AND NOT PRG_BatteryComm.CorvusBMS_Total_Comm_Fault),
	delay11 := T#5s,
	out11 => Warning_CellVolt_LL_Offline,

	(*Low SoC while Offline*)
	in12 := ((minPackSoC < PRG_HMI.SetupBatLimits.SoCTripLL_Offline)
	 			AND NOT PRG_BatteryComm.CorvusBMS_Total_Comm_Fault
	),
	delay12 := T#5s,
	out12 => Warning_SoC_LL_Offline,

	Reset:= PRG_Functions.Reset,
	outCommon =>
);

(*
 * =======================================================================================================================================
 * Offline Protection
 * =======================================================================================================================================
*)

ForceSleepMode := ((minCellTemp < PRG_HMI.SetupBatLimits.CellVoltTripLL_Offline) OR (minPackSoC < PRG_HMI.SetupBatLimits.SoCTripLL_Offline)) AND NOT BatteryCharging;

(*----------------------------------------Find lowest and highest cell voltage----------------------------------------*)

(*Find lowest cell voltage in array*)
FOR i:=1 TO PRG_HMI.setup_Battery_total_nr_of_packs BY 1 DO
	minCellVoltageArray[i] := DINT_TO_REAL(CorvusRead[i].Pack.minCellVoltage);
END_FOR
(*If there are fewer packs than 16, make sure that there are no zeros in the array as we are looking for the lowest number. *)
IF (PRG_HMI.setup_Battery_total_nr_of_packs < 16) THEN
	FOR i:=(PRG_HMI.setup_Battery_total_nr_of_packs+1) TO 16 BY 1 DO
		minCellVoltageArray[i] := 9999;
	END_FOR
END_IF
(*Finally, find the lowest cell voltage and store it*)
minCellVoltage := REAL_TO_INT(ARRAY_MIN(pt := ADR(minCellVoltageArray), size:=SIZEOF(minCellVoltageArray)));

(*Find highest cell voltage in array*)
FOR i:=1 TO PRG_HMI.setup_Battery_total_nr_of_packs BY 1 DO
	maxCellVoltageArray[i] := DINT_TO_REAL(CorvusRead[i].Pack.maxCellVoltage);
END_FOR

(*Finally, find the highest cell voltage and store it*)
maxCellVoltage := REAL_TO_INT(ARRAY_MAX(pt := ADR(maxCellVoltageArray), size:=SIZEOF(maxCellVoltageArray)));

(*--------------------------------------Find lowest and highest cell temperature--------------------------------------*)

(*Find lowest cell temperature in array*)
FOR i:=1 TO PRG_HMI.setup_Battery_total_nr_of_packs BY 1 DO
	minCellTempArray[i] := DINT_TO_REAL(CorvusRead[i].Pack.minCellTemp);
END_FOR
(*If there are fewer packs than 16, make sure that there are no zeros in the array as we are looking for the lowest number. *)
IF (PRG_HMI.setup_Battery_total_nr_of_packs < 16) THEN
	FOR i:=(PRG_HMI.setup_Battery_total_nr_of_packs+1) TO 16 BY 1 DO
		minCellTempArray[i] := 9999;
	END_FOR
END_IF
(*Finally, find the lowest cell temperature and store it*)
minCellTemp := REAL_TO_INT(ARRAY_MIN(pt := ADR(minCellTempArray), size:=SIZEOF(minCellTempArray)));

(*Find highest cell temperature in array*)
FOR i:=1 TO PRG_HMI.setup_Battery_total_nr_of_packs BY 1 DO
	maxCellTempArray[i] := DINT_TO_REAL(CorvusRead[i].Pack.maxCellTemp);
END_FOR

(*Finally, find the highest cell temperature and store it*)
maxCellTemp := REAL_TO_INT(ARRAY_MAX(pt := ADR(maxCellTempArray), size:=SIZEOF(maxCellTempArray)));

(*------------------------------------------Find lowest and highest pack SoC------------------------------------------*)

(*Find lowest pack SoC in array*)
FOR i:=1 TO PRG_HMI.setup_Battery_total_nr_of_packs BY 1 DO
	minPackSoCArray[i] := DINT_TO_REAL(CorvusRead[i].Pack.SOC);
END_FOR
(*If there are fewer packs than 16, make sure that there are no zeros in the array as we are looking for the lowest number. *)
IF (PRG_HMI.setup_Battery_total_nr_of_packs < 16) THEN
	FOR i:=(PRG_HMI.setup_Battery_total_nr_of_packs+1) TO 16 BY 1 DO
		minPackSoCArray[i] := 9999;
	END_FOR
END_IF
(*Finally, find the lowest pack SoC and store it*)
minPackSoC := REAL_TO_INT(ARRAY_MIN(pt := ADR(minPackSoCArray), size:=SIZEOF(minPackSoCArray)));

(*Find highest pack SoC in array*)
FOR i:=1 TO PRG_HMI.setup_Battery_total_nr_of_packs BY 1 DO
	maxPackSoCArray[i] := DINT_TO_REAL(CorvusRead[i].Pack.SOC);
END_FOR

(*Finally, find the highest pack SoC and store it*)
maxPackSoC := REAL_TO_INT(ARRAY_MAX(pt := ADR(maxPackSoCArray), size:=SIZEOF(maxPackSoCArray)));

(*
 * =======================================================================================================================================
 * Check and for faults, warning and prewarnings
 * =======================================================================================================================================
*)

(*Check for any faults*)
batteryCommonFault := (PRG_BatteryComm.CorvusRead[M].theArray.nrOfPackFault <> 0);

(*
 * =======================================================================================================================================
 * Search and Create Common Warnings and Faults from BMS
 * =======================================================================================================================================
*)

FOR i:=1 TO PRG_HMI.setup_Battery_total_nr_of_packs BY 1 DO

	(*---------------------------WARNINGS---------------------------*)

	(*Common Cell Over Voltage Warning*)
	IF (PRG_BatteryComm.CorvusRead[i].FW.SE_overVoltage_Warning) THEN
			Common_SE_overVoltage_Warning_Array[i] := 1*i;
	ELSE	Common_SE_overVoltage_Warning_Array[i] := 0;
	END_IF

	(*Common Cell Under Voltage Warning*)
	IF (PRG_BatteryComm.CorvusRead[i].FW.SE_underVoltage_Warning) THEN
			Common_SE_underVoltage_Warning_Array[i] := 1*i;
	ELSE	Common_SE_underVoltage_Warning_Array[i] := 0;
	END_IF

	(*Common Cell Over Temperature Warning*)
	IF (PRG_BatteryComm.CorvusRead[i].FW.SE_overTemperature_Warning) THEN
			Common_SE_overTemperature_Warning_Array[i] := 1*i;
	ELSE	Common_SE_overTemperature_Warning_Array[i] := 0;
	END_IF

	(*Common Module Communication Warning*)
	IF (PRG_BatteryComm.CorvusRead[i].FW.Module_Communication_Warning) THEN
			Common_Module_Communication_Warning_Array[i] := 1*i;
	ELSE	Common_Module_Communication_Warning_Array[i] := 0;
	END_IF

	(*Common Over Current Warning*)
	IF (PRG_BatteryComm.CorvusRead[i].FW.OverCurrent_Warning) THEN
			Common_OverCurrent_Warning_Array[i] := 1*i;
	ELSE	Common_OverCurrent_Warning_Array[i] := 0;
	END_IF

	(* Common Input Powerloss Warning*)
	IF (PRG_BatteryComm.CorvusRead[i].FW.Input_PowerLoss_Warning) THEN
			Common_Input_PowerLoss_Warning_Array[i] := 1*i;
	ELSE	Common_Input_PowerLoss_Warning_Array[i] := 0;
	END_IF

	(*Common Power Distribution Module Over Temperature Warning*)
	IF (PRG_BatteryComm.CorvusRead[i].FW.PDM_overTemperature_Warning) THEN
			Common_PDM_overTemperature_Warning_Array[i] := 1*i;
	ELSE	Common_PDM_overTemperature_Warning_Array[i] := 0;
	END_IF

	(*Common Coolant Water Leakage Warning*)
	IF (PRG_BatteryComm.CorvusRead[i].FW.CoolantLeak_Warning) THEN
			Common_CoolantLeak_Warning_Array[i] := 1*i;
	ELSE	Common_CoolantLeak_Warning_Array[i] := 0;
	END_IF

	(*---------------------------FAULTS---------------------------*)

	(*Common Cell Over Voltage Fault*)
	IF (PRG_BatteryComm.CorvusRead[i].FW.SE_overVoltage_Fault) THEN
			Common_SE_overVoltage_Fault_Array[i] := 1*i;
	ELSE	Common_SE_overVoltage_Fault_Array[i] := 0;
	END_IF

	(*Common Cell Under Voltage Fault*)
	IF (PRG_BatteryComm.CorvusRead[i].FW.SE_underVoltage_Fault) THEN
			Common_SE_underVoltage_Fault_Array[i] := 1*i;
	ELSE	Common_SE_underVoltage_Fault_Array[i] := 0;
	END_IF

	(*Common Cell Over Temperature Fault*)
	IF (PRG_BatteryComm.CorvusRead[i].FW.SE_overTemperature_Fault) THEN
			Common_SE_overTemperature_Fault_Array[i] := 1*i;
	ELSE	Common_SE_overTemperature_Fault_Array[i] := 0;
	END_IF

	(*Common High Voltage Interlock Loop fault*)
	IF (PRG_BatteryComm.CorvusRead[i].FW.HVIL_Fault) THEN
			Common_HVIL_Fault_Array[i] := 1*i;
	ELSE	Common_HVIL_Fault_Array[i] := 0;
	END_IF

	(*Common Emergency Stop Active Fault*)
	IF (PRG_BatteryComm.CorvusRead[i].FW.E_Stop_Active_Fault) THEN
			Common_E_Stop_Active_Fault_Array[i] := 1*i;
	ELSE	Common_E_Stop_Active_Fault_Array[i] := 0;
	END_IF

	(*Common Safety Shutdown Fault*)
	IF (PRG_BatteryComm.CorvusRead[i].FW.Safety_Shutdown_Fault) THEN
			Common_Safety_Shutdown_Fault_Array[i] := 1*i;
	ELSE	Common_Safety_Shutdown_Fault_Array[i] := 0;
	END_IF

	(*Common Ground Fault*)
	IF (PRG_BatteryComm.CorvusRead[i].FW.Ground_Fault) THEN
			Common_Ground_Fault_Fault_Array[i] := 1*i;
	ELSE	Common_Ground_Fault_Fault_Array[i] := 0;
	END_IF

	(*Common Contactor Fault*)
	IF (PRG_BatteryComm.CorvusRead[i].FW.Contactor_Fault) THEN
			Common_Contactor_Fault_Array[i] := 1*i;
	ELSE	Common_Contactor_Fault_Array[i] := 0;
	END_IF

	(*Common Low Temperature Over Current Fault*)
	IF (PRG_BatteryComm.CorvusRead[i].FW.Low_Temp_OverCurrent_Fault) THEN
			Common_Low_Temp_OverCurrent_Fault_Array[i] := 1*i;
	ELSE	Common_Low_Temp_OverCurrent_Fault_Array[i] := 0;
	END_IF

	(*Common Repeated Over Charge Lockout Fault*)
	IF (PRG_BatteryComm.CorvusRead[i].FW.Repeated_OverCharge_Lockout_Fault) THEN
			Common_Repeated_OverCharge_Lockout_Fault_Array[i] := 1*i;
	ELSE	Common_Repeated_OverCharge_Lockout_Fault_Array[i] := 0;
	END_IF

	(*Common Deep Over Discharge Lockout Fault*)
	IF (PRG_BatteryComm.CorvusRead[i].FW.Deep_OverDischarge_Lockout_Fault) THEN
			Common_Deep_OverDischarge_Lockout_Fault_Array[i] := 1*i;
	ELSE	Common_Deep_OverDischarge_Lockout_Fault_Array[i] := 0;
	END_IF

	(*Common Power Distribution Module Over Temperature Fault*)
	IF (PRG_BatteryComm.CorvusRead[i].FW.PDM_OverTemperature_Fault) THEN
			Common_PDM_OverTemperature_Fault_Array[i] := 1*i;
	ELSE	Common_PDM_OverTemperature_Fault_Array[i] := 0;
	END_IF

	(* Search for any common warning amongst the battery arrays*)
	IF (PRG_BatteryComm.CorvusRead[i].FW.Alarm_status = 2) THEN
			BatteryWarnings_Array[i] := 1*i;
	ELSE	BatteryWarnings_Array[i] := 0;
	END_IF

	(*Search for warnings associated with pre-warnings*)
	IF (PRG_BatteryComm.CorvusRead[i].FW.OverCurrent_Warning OR
	 PRG_BatteryComm.CorvusRead[i].FW.PDM_overTemperature_Warning OR
	 PRG_BatteryComm.CorvusRead[i].FW.SE_overTemperature_Warning OR
	 PRG_BatteryComm.CorvusRead[i].FW.SE_overVoltage_Warning OR
	 PRG_BatteryComm.CorvusRead[i].FW.OverCurrent_Warning OR
	 PRG_BatteryComm.CorvusRead[i].FW.SE_underVoltage_Warning)
	 THEN
			BatteryPreWarnings_Array[i] := 1*i;
	ELSE	BatteryPreWarnings_Array[i] := 0;
	END_IF

END_FOR
(*Find any warning from battery array*)
Common_SE_overVoltage_Warning := 		( ARRAY_MAX(pt := ADR(Common_SE_overVoltage_Warning_Array), 		size := SIZEOF(Common_SE_overVoltage_Warning_Array))   <> 0);
Common_SE_underVoltage_Warning := 		( ARRAY_MAX(pt := ADR(Common_SE_underVoltage_Warning_Array), 		size := SIZEOF(Common_SE_underVoltage_Warning_Array))   <> 0);
Common_SE_overTemperature_Warning := 	( ARRAY_MAX(pt := ADR(Common_SE_overTemperature_Warning_Array), 	size := SIZEOF(Common_SE_overTemperature_Warning_Array))   <> 0);
Common_Module_Communication_Warning := 	( ARRAY_MAX(pt := ADR(Common_Module_Communication_Warning_Array), 	size := SIZEOF(Common_Module_Communication_Warning_Array))   <> 0);
Common_OverCurrent_Warning := 			( ARRAY_MAX(pt := ADR(Common_OverCurrent_Warning_Array), 			size := SIZEOF(Common_OverCurrent_Warning_Array))   <> 0);
Common_Input_PowerLoss_Warning := 		( ARRAY_MAX(pt := ADR(Common_Input_PowerLoss_Warning_Array), 		size := SIZEOF(Common_Input_PowerLoss_Warning_Array))   <> 0);
Common_PDM_overTemperature_Warning := 	( ARRAY_MAX(pt := ADR(Common_PDM_overTemperature_Warning_Array), 	size := SIZEOF(Common_PDM_overTemperature_Warning_Array))   <> 0);
Common_CoolantLeak_Warning := 			( ARRAY_MAX(pt := ADR(Common_CoolantLeak_Warning_Array), 			size := SIZEOF(Common_CoolantLeak_Warning_Array))   <> 0);

(*Find any fault from battery array*)
Common_SE_overVoltage_Fault := 				( ARRAY_MAX(pt := ADR(Common_SE_overVoltage_Fault_Array), 				size := SIZEOF(Common_SE_overVoltage_Fault_Array))   <> 0);
Common_SE_underVoltage_Fault := 			( ARRAY_MAX(pt := ADR(Common_SE_underVoltage_Fault_Array), 				size := SIZEOF(Common_SE_underVoltage_Fault_Array))   <> 0);
Common_SE_overTemperature_Fault := 			( ARRAY_MAX(pt := ADR(Common_SE_overTemperature_Fault_Array), 			size := SIZEOF(Common_SE_overTemperature_Fault_Array))   <> 0);
Common_HVIL_Fault := 						( ARRAY_MAX(pt := ADR(Common_HVIL_Fault_Array), 						size := SIZEOF(Common_HVIL_Fault_Array))   <> 0);
Common_E_Stop_Active_Fault := 				( ARRAY_MAX(pt := ADR(Common_E_Stop_Active_Fault_Array), 				size := SIZEOF(Common_E_Stop_Active_Fault_Array))   <> 0);
Common_Safety_Shutdown_Fault := 			( ARRAY_MAX(pt := ADR(Common_Safety_Shutdown_Fault_Array), 				size := SIZEOF(Common_Safety_Shutdown_Fault_Array))   <> 0);
Common_Ground_Fault_Fault := 				( ARRAY_MAX(pt := ADR(Common_Ground_Fault_Fault_Array), 				size := SIZEOF(Common_Ground_Fault_Fault_Array))   <> 0);
Common_Contactor_Fault := 					( ARRAY_MAX(pt := ADR(Common_Contactor_Fault_Array), 					size := SIZEOF(Common_Contactor_Fault_Array))   <> 0);
Common_Low_Temp_OverCurrent_Fault := 		( ARRAY_MAX(pt := ADR(Common_Low_Temp_OverCurrent_Fault_Array),			size := SIZEOF(Common_Low_Temp_OverCurrent_Fault_Array))   <> 0);
Common_Repeated_OverCharge_Lockout_Fault := ( ARRAY_MAX(pt := ADR(Common_Repeated_OverCharge_Lockout_Fault_Array),	size := SIZEOF(Common_Repeated_OverCharge_Lockout_Fault_Array))   <> 0);
Common_Deep_OverDischarge_Lockout_Fault := 	( ARRAY_MAX(pt := ADR(Common_Deep_OverDischarge_Lockout_Fault_Array), 	size := SIZEOF(Common_Deep_OverDischarge_Lockout_Fault_Array))   <> 0);
Common_PDM_OverTemperature_Fault := 		( ARRAY_MAX(pt := ADR(Common_PDM_OverTemperature_Fault_Array), 			size := SIZEOF(Common_PDM_OverTemperature_Fault_Array))   <> 0);

(*Prewarning*)
batteryPreWarning := 		(ARRAY_MAX(pt := ADR(BatteryPreWarnings_Array), 	size := SIZEOF(BatteryPreWarnings_Array)) <> 0);

(*Common Warning*)
batteryCommonWarning :=		(ARRAY_MAX(pt := ADR(BatteryWarnings_Array), 		size := SIZEOF(BatteryWarnings_Array)) <> 0);

END_PROGRAM
